ABB RobotStudio station: RobotStudio_PickAndPlace.rspag

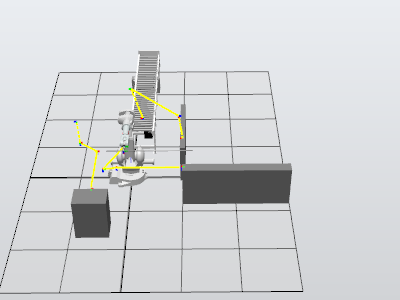
--- station ---
Station Project2 (saved by RobotStudio 23.2.10395.0)
Controller IRB2400_16_150
  mechanical unit ROB_1: IRB2400_16_150__02, 6 joints, base frame (0, 0, 0) mm
Layout (positions relative to the parent item):
  - PinzaGrippe [mechanism] at (0, -940, 1455) mm, rotated rx 0 ry 90 rz -90 deg
      TCP PinzaGrippe at (0, 0, 125) mm
      links: Pinza
  - IRB2400_16_150__02 [mechanism, from %ABB.RobotStudio.Models.IRB2400%\IRB2400_16_150_G_02.rslib] at (0, 0, 0) mm; joint values [-1.5708, 0, 0, 0, 0, 0] (rad or m)
  - Tubo [part] at (1200, -1065, 1455) mm, rotated rx 90 ry 0 rz -90 deg, size 15.9 x 15.9 x 1500 mm
  - SoporteTubo [part] at (0, 1000, 0) mm, size 100 x 1500 x 790 mm
  - Banda ida [part, from %ABB.RobotStudio.Models.Conveyors%\Conveyor Guide 400.rslib] at (0, 3500, 0) mm, rotated rx 0 ry 0 rz -90 deg
  - Doblado [part], size 2000 x 200 x 800 mm
  - CorteBocaPez [part] at (100, -100, 0) mm, size 600 x 400 x 800 mm
  - Sistema de coordenadas_1 [frame] at (0, 0, 100) mm
Attachment: PinzaGrippe is attached to IRB2400_16_150__02 / Link6
Attachment: Tubo is attached to PinzaGrippe / Pinza
Targets, tools, work objects and paths stored in the station and not in the controller backup, written as RAPID:
! task T_ROB1
MODULE CalibData
  PERS tooldata PinzaGrippe:=[TRUE,[[0,0,125],[1,0,0,0]],[1,[0,0,1],[1,0,0,0],0,0,0]];
ENDMODULE

! task T_ROB1
MODULE Module1
  CONST robtarget BandaI:=[[1000,200,800],[0,0,1,0],[-1,0,-1,0],[9E+09,9E+09,9E+09,9E+09,9E+09,9E+09]];
  CONST jointtarget BandaI_Home:=[[0,0,0,0,0,0],[9E+09,9E+09,9E+09,9E+09,9E+09,9E+09]];
  CONST robtarget BandaO:=[[200,900,800],[0,0,1,0],[0,0,0,0],[9E+09,9E+09,9E+09,9E+09,9E+09,9E+09]];
  CONST robtarget DobladoPos:=[[1000,-700,800],[0,0.707106781,0.707106781,0],[-1,0,0,0],[9E+09,9E+09,9E+09,9E+09,9E+09,9E+09]];
  CONST robtarget DobladoAcerL:=[[-200,-700,800],[0,0.707106781,0.707106781,0],[-2,0,-1,0],[9E+09,9E+09,9E+09,9E+09,9E+09,9E+09]];
  CONST robtarget DobladoAc:=[[-400,-1000,1000],[0,0.707106781,0.707106781,0],[-2,0,-1,0],[9E+09,9E+09,9E+09,9E+09,9E+09,9E+09]];
  CONST jointtarget BandaO_Home:=[[90,0,0,0,0,0],[9E+09,9E+09,9E+09,9E+09,9E+09,9E+09]];
  CONST jointtarget Dobladora_Home:=[[-90,0,0,0,0,0],[9E+09,9E+09,9E+09,9E+09,9E+09,9E+09]];
  CONST robtarget Corte_Extremo:=[[-600,-1300,800],[0,1,0,0],[-2,0,0,0],[9E+09,9E+09,9E+09,9E+09,9E+09,9E+09]];
  CONST robtarget Corte_Entrada:=[[-600,-200,800],[0,1,0,0],[-2,0,0,0],[9E+09,9E+09,9E+09,9E+09,9E+09,9E+09]];
  CONST robtarget Corte_Ac:=[[-900,-200,1000],[0,1,0,0],[-2,0,0,0],[9E+09,9E+09,9E+09,9E+09,9E+09,9E+09]];
  CONST jointtarget CorteBocaPez:=[[-170,0,0,0,0,0],[9E+09,9E+09,9E+09,9E+09,9E+09,9E+09]];
  PROC ColocarDobladora()
    MoveAbsJ Dobladora_Home,v1000,z100,PinzaGrippe\WObj:=wobj0;
    MoveJ DobladoAc,v1000,z100,PinzaGrippe\WObj:=wobj0;
    MoveL DobladoAcerL,v1000,z100,PinzaGrippe\WObj:=wobj0;
    MoveL DobladoPos,v1000,z100,PinzaGrippe\WObj:=wobj0;
    MoveL DobladoAcerL,v1000,z100,PinzaGrippe\WObj:=wobj0;
    MoveJ DobladoAc,v1000,z100,PinzaGrippe\WObj:=wobj0;
    MoveAbsJ Dobladora_Home,v1000,z100,PinzaGrippe\WObj:=wobj0;
  ENDPROC
  PROC Verificacion()
    MoveAbsJ BandaI_Home,v1000,z100,PinzaGrippe\WObj:=wobj0;
    MoveJ BandaI,v1000,z100,PinzaGrippe\WObj:=wobj0;
    MoveAbsJ BandaI_Home,v1000,z100,PinzaGrippe\WObj:=wobj0;
    MoveAbsJ BandaO_Home,v1000,z100,PinzaGrippe\WObj:=wobj0;
    MoveJ BandaO,v1000,z100,PinzaGrippe\WObj:=wobj0;
    MoveAbsJ BandaO_Home,v1000,z100,PinzaGrippe\WObj:=wobj0;
    MoveAbsJ BandaI_Home,v1000,z100,PinzaGrippe\WObj:=wobj0;
  ENDPROC
  PROC Corte()
    MoveAbsJ CorteBocaPez,v1000,z100,PinzaGrippe\WObj:=wobj0;
    MoveJ Corte_Ac,v1000,z100,PinzaGrippe\WObj:=wobj0;
    MoveL Corte_Entrada,v1000,z100,PinzaGrippe\WObj:=wobj0;
    MoveL Corte_Extremo,v1000,z100,PinzaGrippe\WObj:=wobj0;
    MoveL Corte_Entrada,v1000,z100,PinzaGrippe\WObj:=wobj0;
    MoveJ Corte_Ac,v1000,z100,PinzaGrippe\WObj:=wobj0;
    MoveAbsJ CorteBocaPez,v1000,z100,PinzaGrippe\WObj:=wobj0;
  ENDPROC
ENDMODULE


--- Controller Data/IRB2400_16_150/RAPID/TASK1/PROGMOD/Module1.mod ---
MODULE Module1
    !***********************************************************
    !
    ! M?dulo:  Module1
    !
    ! Descripción:
    !   <Introduzca la descripción aquí>
    !
    ! Autor: Andrago
    !
    ! Versión: 1.0
    !
    !***********************************************************


    !***********************************************************
    !
    ! Procedimiento Main
    !
    !   Este es el punto de entrada de su programa
    !
    !***********************************************************
    PROC main()
        !Add your code here
    ENDPROC
ENDMODULE
